(* PLC project SafeLOGIC-1, BrAutomation SafeDESIGNER  4.3.4.4 *)
(* stored: companyURL http://www.br-automation.com, creationDateTime Fri Jun 25 07:55:22 2021 *)

PROGRAM Main
  VAR  (* added by the conversion: wires and edge detectors of the diagram *)
    _SAFEBOOL_TO_BOOL22_OUT : BOOL;
  END_VAR

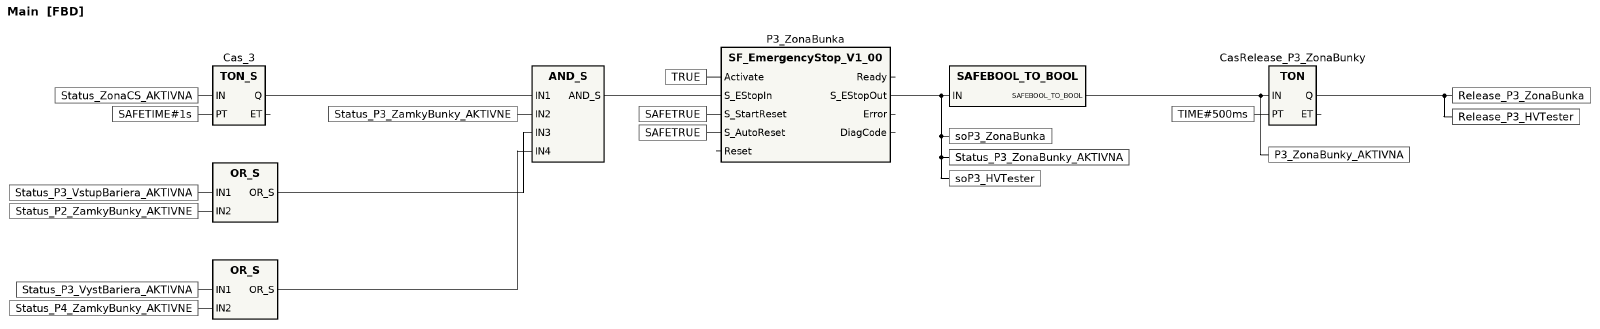
(* FBD diagram, written out as Structured Text *)
Cas_3(IN := Status_ZonaCS_AKTIVNA, PT := SAFETIME#1s);
P3_ZonaBunka(Activate := TRUE, S_EStopIn := AND_S(Cas_3.Q, Status_P3_ZamkyBunky_AKTIVNE, OR_S(Status_P3_VstupBariera_AKTIVNA, Status_P2_ZamkyBunky_AKTIVNE), OR_S(Status_P3_VystBariera_AKTIVNA, Status_P4_ZamkyBunky_AKTIVNE)), S_StartReset := SAFETRUE, S_AutoReset := SAFETRUE);
soP3_ZonaBunka := P3_ZonaBunka.S_EStopOut;
soP3_HVTester := P3_ZonaBunka.S_EStopOut;
Status_P3_ZonaBunky_AKTIVNA := P3_ZonaBunka.S_EStopOut;
_SAFEBOOL_TO_BOOL22_OUT := SAFEBOOL_TO_BOOL(P3_ZonaBunka.S_EStopOut);
P3_ZonaBunky_AKTIVNA := _SAFEBOOL_TO_BOOL22_OUT;
CasRelease_P3_ZonaBunky(IN := _SAFEBOOL_TO_BOOL22_OUT, PT := TIME#500ms);
Release_P3_ZonaBunka := CasRelease_P3_ZonaBunky.Q;
Release_P3_HVTester := CasRelease_P3_ZonaBunky.Q;
END_PROGRAM
